// TIA Portal V20 export
// export: Created 2026-09-14T11:29:00.919355Z, ExportSetting None, DisplayName Totally Integrated Automation Portal, DisplayVersion V20, DisplayName TIA Portal Openness, DisplayVersion V20, DisplayName TIA Portal Version Control Interface, DisplayVersion V20, DisplayName STEP 7 Professional, DisplayVersion V20, DisplayName STEP 7 Safety, DisplayVersion V20, DisplayName WinCC Basic/Comfort/Advanced, DisplayVersion V20, DisplayName WinCC Unified, DisplayVersion V20
TYPE "LMQTT_typeConnectFlags"
   STRUCT
      cleanSession : Bool;   // When TRUE, all data from a previous session will be deleted
      will : Bool;   // When TRUE, activates the last will and testament function
      willQoS1 : Bool;   // When TRUE, the QoS has level 1 for the last will
      willQoS2 : Bool;   // When TRUE, the QoS has level 2 for the last will
      willRetain : Bool;   // When TRUE, the last will is stored at the broker after its been sent
      password : Bool;   // When TRUE, the MQTT broker requires a login (name and password) of the client
      userName : Bool;   // When TRUE, the MQTT broker requires a login (name and password) of the client
   END_STRUCT;
END_TYPE
